FUNCTION_BLOCK FB_ADD
VAR_INPUT
	in1,in2:INT;
END_VAR
VAR_OUTPUT
	out:INT;
END_VAR
VAR
END_VAR

out:=in1+in2;

END_FUNCTION_BLOCK

(* stored: Version 1.1.0.1, ProductVersion 3.1.4024.3
   POU FB_ADD: Id {cd57e488-1c71-4eea-a2e6-5d1a178aab23}, SpecialFunc None *)
